{attribute 'no_explicit_call' := 'do not call this function block directly'} 
FUNCTION_BLOCK DeleteFile EXTENDS ToolkitObject IMPLEMENTS IAction
VAR
	{attribute 'OPC.UA.DA' := '0'}
	_ClassName : STRING := __POUNAME();

	{attribute 'OPC.UA.DA' := '0'}
    _Delete : Tc2_System.FB_FileDelete;
	
	{attribute 'OPC.UA.DA' := '0'}
	_NeedStart : BOOL;
	{attribute 'OPC.UA.DA' := '0'}
	_Done : BOOL;
END_VAR

{attribute 'monitoring' := 'call'}
{attribute 'OPC.UA.DA.Property' := '1'}
{attribute 'OPC.UA.DA' := '1'}
PROPERTY AmsNetId : Tc2_System.T_AmsNetID
GET
AmsNetId := _Delete.sNetId;
END_GET
SET
_Delete.sNetId := AmsNetId;
END_SET
END_PROPERTY

{attribute 'monitoring' := 'call'}
{attribute 'OPC.UA.DA.Property' := '1'}
{attribute 'OPC.UA.DA.Access' := '1'}
PROPERTY Busy : BOOL
GET
Busy := _NeedStart OR_ELSE _Delete.bBusy;
END_GET
END_PROPERTY

{attribute 'monitoring' := 'call'}
PROPERTY ClassName : STRING
GET
ClassName := _ClassName;
END_GET
END_PROPERTY

{attribute 'monitoring' := 'call'}
{attribute 'OPC.UA.DA.Property' := '1'}
{attribute 'OPC.UA.DA.Access' := '1'}
PROPERTY Done : BOOL
GET
Done := _Done;
END_GET
END_PROPERTY

{attribute 'monitoring' := 'call'}
{attribute 'OPC.UA.DA.Property' := '1'}
{attribute 'OPC.UA.DA.Access' := '1'}
PROPERTY Error : BOOL
GET
Error := _Delete.bError;
END_GET
END_PROPERTY

METHOD Execute
VAR
	message : ERROR_MESSAGE;
END_VAR
IF _NeedStart OR_ELSE _Delete.bBusy THEN
	_Delete(bExecute := TRUE);
	_NeedStart := FALSE;
	
	IF _Delete.bError THEN
		message := "An error occurred while creating the file '";
		WStringHelper.Append2(message, TO_WSTRING(_Delete.sPathName), "'");	
		_LastException.Configure(message, __POUNAME(), ClassName, CurrentNamespace.Name, __POSITION(), _Delete.nErrId).Throw();
	ELSIF NOT _Delete.bBusy THEN
		_Done := TRUE;
	END_IF
END_IF
END_METHOD

{attribute 'monitoring' := 'call'}
{attribute 'OPC.UA.DA.Property' := '1'}
{attribute 'OPC.UA.DA.Access' := '1'}
PROPERTY LastException : REFERENCE TO Exception
GET
LastException REF= _LastException;
END_GET
END_PROPERTY

{attribute 'monitoring' := 'call'}
{attribute 'OPC.UA.DA.Property' := '1'}
{attribute 'OPC.UA.DA' := '1'}
PROPERTY PathType : Tc2_System.E_OpenPath
GET
PathType := _Delete.ePath;
END_GET
SET
_Delete.ePath := PathType;
END_SET
END_PROPERTY

METHOD Start
VAR_INPUT
	filePath : Tc2_System.T_MaxString;
END_VAR
_NeedStart := TRUE;
_Done := FALSE;
_Delete.sPathName := filePath;

_LastException.Clear();
END_METHOD

{attribute 'monitoring' := 'call'}
{attribute 'OPC.UA.DA.Property' := '1'}
{attribute 'OPC.UA.DA' := '1'}
PROPERTY Timeout : TIME
GET
Timeout := _Delete.tTimeout;
END_GET
SET
_Delete.tTimeout := Timeout;
END_SET
END_PROPERTY

END_FUNCTION_BLOCK

(* stored: Version 1.1.0.1
   POU DeleteFile: Id {76565d63-59cb-438d-9547-03e346761d4d}, SpecialFunc None
   Property AmsNetId: Id {db7ca382-eeba-493b-9ca5-d1bd68de1a30}
   Get Get: Id {20505ad8-7d29-4835-95fa-3f92abc311c9}
   Set Set: Id {fc6f2a4f-a739-473b-a3f8-09da3e29f4b4}
   Property Busy: Id {15729b8e-6317-4e62-9f1f-832a4247abcf}
   Get Get: Id {0d0a0b86-6257-46e4-87c2-42a273d47e7e}
   Property ClassName: Id {d3939381-7f4e-462e-bead-9da89ec8fc63}
   Get Get: Id {648bbaeb-2257-434e-a70a-0157df4a8be1}
   Property Done: Id {89305253-c30c-4247-ab1b-7be8187a9f57}
   Get Get: Id {35dfdffd-5bfe-48bf-a9ee-1431e0475117}
   Property Error: Id {7fb63d6b-be79-4e0a-891f-7fe516c23a8d}
   Get Get: Id {0fe004e6-855f-4c47-bca3-cc592b5c5f72}
   Method Execute: Id {89d7f19a-8d96-4dce-a596-a9e3243a8010}
   Property LastException: Id {a907e474-ef8c-428a-b91b-40d37f3d5eec}
   Get Get: Id {c6d589d7-d90f-4aee-ad72-a968b81fbdb1}
   Property PathType: Id {24f35cd6-3bdd-48a7-ba3f-8d9951259501}
   Get Get: Id {de876974-58e7-4cb4-a64b-0e39015e32ce}
   Set Set: Id {e1ecf7f0-64d9-4217-b21e-5d27aca361a0}
   Method Start: Id {59ca7d6b-c42a-44f6-a7af-5bd06c0862ef}
   Property Timeout: Id {c3e15cad-6f39-46dc-b7d3-d1ade209a2b7}
   Get Get: Id {07cd4b08-8cff-4e6d-b487-3a7f25030a7b}
   Set Set: Id {b6c8adff-556b-4f72-a425-0b9744d4f382} *)
